// TIA Portal V19 export
DATA_BLOCK "ControlNodes"   // DB47
// stored: Access Published, MemoryReserve 100, Namespace Unit2.EM4
   VAR
      em { ExternalWritable := 'False'} : "LAF_typeEmControlNode";
      jobs { ExternalWritable := 'False'} : "LAF_typeJobs";
      sequence { ExternalWritable := 'False'} : "LAF_typeSequence";
      cm1AxisControl : "LBC_typeAxisSimpleControlNode_1";
      cm2AxisControl { S7_SetPoint := 'True'} : "LBC_typeAxisSimpleControlNode_1";
      cm3AxisControl { S7_SetPoint := 'True'} : "LBC_typeAxisSimpleControlNode_1";
      cm4Cylinder { S7_SetPoint := 'True'} : "LBC_Simple_typeTwoWayActuatorControlNode";
      cm5Cylinder { S7_SetPoint := 'True'} : "LBC_Simple_typeTwoWayActuatorControlNode";
      cm6Cylinder { S7_SetPoint := 'True'} : "LBC_Simple_typeTwoWayActuatorControlNode";
      cm7Cylinder { S7_SetPoint := 'True'} : "LBC_Simple_typeTwoWayActuatorControlNode";
      cm8SignalTM { S7_SetPoint := 'True'} : "LEXCHANGETRAY_typeHandlingXyzIoSignalControlNode";
      stepCondition { S7_SetPoint := 'True'} : "LEXCHANGETRAY_typeConstraintRollerTranserfCondition";
   END_VAR
BEGIN
   em.status.enabled := true;
END_DATA_BLOCK
